//---------------------------------------------------------------------------------------------------------------
//
//  HAUD 2026.01.16
//
//  - ExternControl
//
//    - cyclic call to simulation class which handshakes the XtsStations in XtsTransport PLC
//
//---------------------------------------------------------------------------------------------------------------
PROGRAM MAIN_APP
VAR
  eInitXtsTransport   AT %I*    : e_progress;
  eInit                         : E_PROGRESS;   // application startup state info

  nProcess          : UINT;

  bNext             : BOOL := TRUE;
  bEnter            : BOOL := TRUE;
  bLeave            : BOOL := TRUE;

  tProcess          : ARRAY[1..MAX_PROCESS] OF TIME;

  eMtrState,
  eMsgState         : E_MESSAGE_STATE;
  eMtrProgress,
  eMsgProgress      : e_progress;
  stMsg             : ST_Message;
  //-------------------------------------------------------------------------------------------------------------
  tIdleWriteApplication   : TIME := T#5S;
  tIdleWriteMetric        : TIME := T#5S;
  tonIdleWriteApplication : Tc2_Standard.TON;
  tonIdleWriteMetric      : Tc2_Standard.TON;
  //-------------------------------------------------------------------------------------------------------------
END_VAR

//#################################################################################################################
// Local time; used for timestamps
//#################################################################################################################
GVL_MSG_XTS.fbLocalTime();
GVL_MSG_XTS.sLocalTime                                      := GVL_MSG_XTS.fbLocalTime.LocalTimeString;
GVL_MSG_XTS.dtLocalTime                                     := GVL_MSG_XTS.fbLocalTime.LocalTime;
//#################################################################################################################
//#################################################################################################################
//-----------------------------------------------------------------------------------------------------------------
//-----------------------------------------------------------------------------------------------------------------
// check for MAIN.eInit
//  - wait for fb_TransportUnit to be fully started up
//-----------------------------------------------------------------------------------------------------------------
IF NOT (eInitXtsTransport = E_PROGRESS.PROGRESS_DONE) THEN eInit   := E_PROGRESS.PROGRESS_INVALID; RETURN; END_IF
//-----------------------------------------------------------------------------------------------------------------
//-----------------------------------------------------------------------------------------------------------------
//-----------------------------------------------------------------------------------------------------------------
// /assign dataflow
//-----------------------------------------------------------------------------------------------------------------
FOR nProcess := 1 TO MAX_PROCESS
DO
  GVL_APPLICATION.Simulation[nProcess].ProcessId            := nProcess;
  GVL_APPLICATION.Simulation[nProcess].StationCtrl          := ADR(GVL_XTS.StationCtrl);
  GVL_APPLICATION.Simulation[nProcess].StationState         := ADR(GVL_XTS.StationState);

  GVL_APPLICATION.Simulation[nProcess].ProcessTime          := tProcess[nProcess];
  GVL_APPLICATION.Simulation[nProcess].MessageLevel         := GVL_MSG_XTS.MessageLevel;
END_FOR
//-----------------------------------------------------------------------------------------------------------------
//-----------------------------------------------------------------------------------------------------------------
Init();
//-----------------------------------------------------------------------------------------------------------------
//-----------------------------------------------------------------------------------------------------------------
// react to operation modes
//-----------------------------------------------------------------------------------------------------------------
//-----------------------------------------------------------------------------------------------------------------
CASE GVL_XTS.XtsTransportCtrl.Cmd
OF
  E_XTS_TRANSPORT_CTRL.CMD_INIT,
  E_XTS_TRANSPORT_CTRL.CMD_GROUP_CLEAR:

    FOR nProcess := 1 TO MAX_PROCESS
    DO
      GVL_APPLICATION.Simulation[nProcess].Init(); // clearing of XtsStations and Simulation
    END_FOR
END_CASE

CASE (GVL_XTS.XtsTransportState.State MOD E_PROGRESS.PROGRESS_DONE)
OF
  E_XTS_TRANSPORT_STATE.TRANSPORT_INIT,
  E_XTS_TRANSPORT_STATE.TRANSPORT_GROUP_CLEAR:
    FOR nProcess := 1 TO MAX_PROCESS
    DO
      GVL_APPLICATION.Simulation[nProcess].Disable(); // switch off XtsStations and clear Simulation

      GVL_APPLICATION.Simulation[nProcess].EnableProcess    := 0;
      GVL_APPLICATION.Simulation[nProcess].MoverEnter       := FALSE;
      GVL_APPLICATION.Simulation[nProcess].MoverOut         := FALSE;

      GVL_APPLICATION.Simulation[nProcess].Cycle();
    END_FOR

  E_XTS_TRANSPORT_STATE.TRANSPORT_START,
  E_XTS_TRANSPORT_STATE.TRANSPORT_RESTART:

    FOR nProcess := 1 TO MAX_PROCESS
    DO
      GVL_APPLICATION.Simulation[nProcess].Next(bNext);
      GVL_APPLICATION.Simulation[nProcess].Cycle();
    END_FOR
ELSE
  CASE (GVL_XTS.XtsTransportState.State MOD E_PROGRESS.PROGRESS_WORKING)
  OF
  E_XTS_TRANSPORT_STATE.TRANSPORT_START,
  E_XTS_TRANSPORT_STATE.TRANSPORT_RESTART:
    FOR nProcess := 1 TO MAX_PROCESS
    DO
      IF (GVL_APPLICATION.Simulation[nProcess].StationCount > 0)
      THEN
        GVL_APPLICATION.Simulation[nProcess].EnableProcess  := TO_DWORD(EXPT(2,GVL_APPLICATION.Simulation[nProcess].StationCount))-1;
        GVL_APPLICATION.Simulation[nProcess].MoverEnter     := TRUE;
        GVL_APPLICATION.Simulation[nProcess].MoverOut       := TRUE;

      END_IF

      GVL_APPLICATION.Simulation[nProcess].Next(bNext);
      GVL_APPLICATION.Simulation[nProcess].Cycle();
    END_FOR
  END_CASE
END_CASE
//-----------------------------------------------------------------------------------------------------------------
//-----------------------------------------------------------------------------------------------------------------
//#################################################################################################################
// /logging
//#################################################################################################################
GVL_MSG_XTS.ApplicationMessageData.Ctrl                         REF= GVL_MSG_XTS.ApplicationMessageCtrl;
GVL_MSG_XTS.ApplicationMessageData.State                        REF= GVL_MSG_XTS.ApplicationMessageState;

GVL_MSG_XTS.ApplicationMessageData.MessageIndex                 REF= GVL_MSG_XTS.MessageApplicationIndex;
GVL_MSG_XTS.ApplicationMessageData.ErrorIndex                   REF= GVL_MSG_XTS.MessageApplicationError;

GVL_MSG_XTS.ApplicationMessageData.DirRoot                      :=   ADR(GVL_MSG_XTS.LOG_DIR);
GVL_MSG_XTS.ApplicationMessageData.FileRoot                     :=   ADR(GVL_MSG_XTS.LOG_FILE_APP);
GVL_MSG_XTS.ApplicationMessageData.MsgList                      :=   ADR(GVL_MSG_XTS.ApplicationMessages);
GVL_MSG_XTS.ApplicationMessageData.LocalTime                    :=   ADR(GVL_MSG_XTS.dtLocalTime);

GVL_MSG_XTS.ApplicationMessageData();

eMsgState                                   := f_GetState   (GVL_MSG_XTS.ApplicationMessageState.State);
eMsgProgress                                := f_GetProgress(GVL_MSG_XTS.ApplicationMessageState.State);


CASE eMsgState
OF
  E_MESSAGE_STATE.MSG_STATE_NULL:
    CASE eMsgProgress
    OF
      E_PROGRESS.PROGRESS_INVALID:
        IF (GVL_MSG_XTS.MessageApplicationIndex > GVL_MSG_XTS.MAX_MESSAGE/100) OR
           (GVL_MSG_XTS.MessageApplicationError > 0)
        THEN
          GVL_MSG_XTS.ApplicationMessageCtrl.Cmd  := E_MESSAGE_CTRL.MSG_CTRL_WRITE;
        ELSE
          tonIdleWriteApplication(IN := TRUE, PT:= tIdleWriteApplication);
          IF (tonIdleWriteApplication.Q)
          THEN
            GVL_MSG_XTS.TransportMessageCtrl.Cmd    := E_MESSAGE_CTRL.MSG_CTRL_WRITE;
          END_IF
        END_IF
    END_CASE

  E_MESSAGE_STATE.MSG_STATE_WRITE:
    CASE eMsgProgress
    OF
      E_PROGRESS.PROGRESS_ERROR,
      E_PROGRESS.PROGRESS_DONE:
        tonIdleWriteApplication(IN := FALSE, PT:= tIdleWriteApplication);
        GVL_MSG_XTS.ApplicationMessageCtrl.Cmd    := E_MESSAGE_CTRL.MSG_CTRL_NULL;
    END_CASE

ELSE
    CASE eMsgProgress
    OF
      E_PROGRESS.PROGRESS_DONE:
        GVL_MSG_XTS.ApplicationMessageCtrl.Cmd    := E_MESSAGE_CTRL.MSG_CTRL_NULL;
    END_CASE
END_CASE
//#################################################################################################################
// logging/
//#################################################################################################################
//#################################################################################################################
//  /Transport Metrics
//#################################################################################################################
GVL_MSG_XTS.MetricsMessageData.Ctrl                             REF= GVL_MSG_XTS.MetricsMessageCtrl;
GVL_MSG_XTS.MetricsMessageData.State                            REF= GVL_MSG_XTS.MetricsMessageState;

GVL_MSG_XTS.MetricsMessageData.MessageIndex                     REF= GVL_MSG_XTS.MessageMetricsIndex;
GVL_MSG_XTS.MetricsMessageData.ErrorIndex                       REF= GVL_MSG_XTS.MessageMetricsError;

GVL_MSG_XTS.MetricsMessageData.DirRoot                          :=   ADR(GVL_MSG_XTS.LOG_DIR);
GVL_MSG_XTS.MetricsMessageData.FileRoot                         :=   ADR(GVL_MSG_XTS.LOG_FILE_METRIC);
GVL_MSG_XTS.MetricsMessageData.MsgList                          :=   ADR(GVL_MSG_XTS.MetricsMessages);
GVL_MSG_XTS.MetricsMessageData.LocalTime                        :=   ADR(GVL_MSG_XTS.dtLocalTime);

GVL_MSG_XTS.MetricsMessageData();

eMtrState                                   := f_GetState   (GVL_MSG_XTS.MetricsMessageState.State);
eMtrProgress                                := f_GetProgress(GVL_MSG_XTS.MetricsMessageState.State);

CASE eMtrState
OF
  E_MESSAGE_STATE.MSG_STATE_NULL:
    CASE eMtrProgress
    OF
      E_PROGRESS.PROGRESS_INVALID:
        IF (GVL_MSG_XTS.MessageMetricsIndex > GVL_MSG_XTS.MAX_MESSAGE/100) OR
           (GVL_MSG_XTS.MessageMetricsError > 0)
        THEN
          GVL_MSG_XTS.MetricsMessageCtrl.Cmd      := E_MESSAGE_CTRL.MSG_CTRL_WRITE;
        ELSE
          tonIdleWriteMetric(IN := TRUE, PT:= tIdleWriteMetric);
          IF (tonIdleWriteMetric.Q)
          THEN
            GVL_MSG_XTS.TransportMessageCtrl.Cmd    := E_MESSAGE_CTRL.MSG_CTRL_WRITE;
          END_IF
        END_IF
    END_CASE

  E_MESSAGE_STATE.MSG_STATE_WRITE:
    CASE eMtrProgress
    OF
      E_PROGRESS.PROGRESS_ERROR,
      E_PROGRESS.PROGRESS_DONE:
        tonIdleWriteMetric(IN := FALSE, PT:= tIdleWriteMetric);
        GVL_MSG_XTS.MetricsMessageCtrl.Cmd        := E_MESSAGE_CTRL.MSG_CTRL_NULL;
    END_CASE
ELSE
    CASE eMtrProgress
    OF
      E_PROGRESS.PROGRESS_DONE:
        GVL_MSG_XTS.MetricsMessageCtrl.Cmd        := E_MESSAGE_CTRL.MSG_CTRL_NULL;
    END_CASE
END_CASE
//#################################################################################################################
//  Transport Metrics/
//#################################################################################################################
//#################################################################################################################
//#################################################################################################################

ACTION Init:
CASE eInit
OF
  E_PROGRESS.PROGRESS_INVALID:          // startup procedure for your application
    GVL_MSG_XTS.TransportMessageCtrl.Cmd                  := E_MESSAGE_CTRL.MSG_CTRL_NULL;
    GVL_MSG_XTS.MetricsMessageCtrl.Cmd                    := E_MESSAGE_CTRL.MSG_CTRL_NULL;

    FOR nProcess := 1 TO MAX_PROCESS
    DO
      GVL_MSG_XTS.MessageLevelProcess[nProcess]           := GVL_MSG_XTS.MessageLevel;

      GVL_APPLICATION.Simulation[nProcess].MessageLevel   := GVL_MSG_XTS.MessageLevelProcess[nProcess];
    END_FOR
    eInit                               := E_PROGRESS.PROGRESS_INIT;


  E_PROGRESS.PROGRESS_INIT:
      nProcess                                        := 1;
      tProcess[nProcess]                              := T#750MS;

      GVL_APPLICATION.Simulation[nProcess].StationFirst  := 1;
      GVL_APPLICATION.Simulation[nProcess].StationLast   := 16;

      GVL_APPLICATION.Simulation[nProcess].TargetFirst   := 20;
      GVL_APPLICATION.Simulation[nProcess].TargetLast    := 35;
      GVL_APPLICATION.Simulation[nProcess].TargetMask    := 2#0001; // mask for target station

      GVL_APPLICATION.Simulation[nProcess].CheckRangeLow := 1750.0;
      GVL_APPLICATION.Simulation[nProcess].CheckRangeHigh:= 2100.0;

      //---------------------------------------------------------

      // 2

      //---------------------------------------------------------
      nProcess                                        := 3;
      tProcess[nProcess]                              := T#1250MS;

      GVL_APPLICATION.Simulation[nProcess].StationFirst  := 20;
      GVL_APPLICATION.Simulation[nProcess].StationLast   := 35;

      GVL_APPLICATION.Simulation[nProcess].TargetFirst   := 37;
      GVL_APPLICATION.Simulation[nProcess].TargetLast    := 37;
      GVL_APPLICATION.Simulation[nProcess].TargetMask    := 2#0001; // mask for target station

      GVL_APPLICATION.Simulation[nProcess].CheckRangeLow := 4500.0;
      GVL_APPLICATION.Simulation[nProcess].CheckRangeHigh:= 5100.0;

      //---------------------------------------------------------
      nProcess                                        := 4;
      tProcess[nProcess]                              := T#0MS;

      GVL_APPLICATION.Simulation[nProcess].StationFirst  := 37;
      GVL_APPLICATION.Simulation[nProcess].StationLast   := 37;

      GVL_APPLICATION.Simulation[nProcess].TargetFirst   := 45;
      GVL_APPLICATION.Simulation[nProcess].TargetLast    := 52;
      GVL_APPLICATION.Simulation[nProcess].TargetMask    := 2#0001; // mask for target station

      GVL_APPLICATION.Simulation[nProcess].CheckRangeLow := 7450.0;
      GVL_APPLICATION.Simulation[nProcess].CheckRangeHigh:= 7600.0;

      //---------------------------------------------------------
      nProcess                                        := 5;
      tProcess[nProcess]                              := T#500MS;

      GVL_APPLICATION.Simulation[nProcess].StationFirst  := 45;
      GVL_APPLICATION.Simulation[nProcess].StationLast   := 52;

      GVL_APPLICATION.Simulation[nProcess].TargetFirst   := 58;
      GVL_APPLICATION.Simulation[nProcess].TargetLast    := 69;
      GVL_APPLICATION.Simulation[nProcess].TargetMask    := 2#0001; // mask for target station

      GVL_APPLICATION.Simulation[nProcess].CheckRangeLow := 6600.0;
      GVL_APPLICATION.Simulation[nProcess].CheckRangeHigh:= 8350.0;

      //---------------------------------------------------------
      nProcess                                        := 6;
      tProcess[nProcess]                              := T#500MS;

      GVL_APPLICATION.Simulation[nProcess].StationFirst  := 58;
      GVL_APPLICATION.Simulation[nProcess].StationLast   := 69;

      GVL_APPLICATION.Simulation[nProcess].TargetFirst   := 70;
      GVL_APPLICATION.Simulation[nProcess].TargetLast    := 81;
      GVL_APPLICATION.Simulation[nProcess].TargetMask    := 2#0001; // mask for target station

      GVL_APPLICATION.Simulation[nProcess].CheckRangeLow := 8750.0;
      GVL_APPLICATION.Simulation[nProcess].CheckRangeHigh:= 9600.0;

      //---------------------------------------------------------
      nProcess                                        := 7;
      tProcess[nProcess]                              := T#500MS;

      GVL_APPLICATION.Simulation[nProcess].StationFirst  := 70;
      GVL_APPLICATION.Simulation[nProcess].StationLast   := 81;

      GVL_APPLICATION.Simulation[nProcess].TargetFirst   := 82;
      GVL_APPLICATION.Simulation[nProcess].TargetLast    := 91;
      GVL_APPLICATION.Simulation[nProcess].TargetMask    := 2#0001; // mask for target station

      GVL_APPLICATION.Simulation[nProcess].CheckRangeLow := 10900.0;
      GVL_APPLICATION.Simulation[nProcess].CheckRangeHigh:= 11600.0;

      //---------------------------------------------------------
      nProcess                                        := 8;
      tProcess[nProcess]                              := T#500MS;

      GVL_APPLICATION.Simulation[nProcess].StationFirst  := 82;
      GVL_APPLICATION.Simulation[nProcess].StationLast   := 91;

      GVL_APPLICATION.Simulation[nProcess].TargetFirst   := 92;
      GVL_APPLICATION.Simulation[nProcess].TargetLast    := 99;
      GVL_APPLICATION.Simulation[nProcess].TargetMask    := 2#0001; // mask for target station

      GVL_APPLICATION.Simulation[nProcess].CheckRangeLow := 12550.0;
      GVL_APPLICATION.Simulation[nProcess].CheckRangeHigh:= 12900.0;

      //---------------------------------------------------------
      nProcess                                        := 9;
      tProcess[nProcess]                              := T#500MS;

      GVL_APPLICATION.Simulation[nProcess].StationFirst  := 92;
      GVL_APPLICATION.Simulation[nProcess].StationLast   := 99;

      GVL_APPLICATION.Simulation[nProcess].TargetFirst   := 118;
      GVL_APPLICATION.Simulation[nProcess].TargetLast    := 118;
      GVL_APPLICATION.Simulation[nProcess].TargetMask    := 2#0001; // mask for target station

      GVL_APPLICATION.Simulation[nProcess].CheckRangeLow := 13600.0;
      GVL_APPLICATION.Simulation[nProcess].CheckRangeHigh:= 14600.0;

      //---------------------------------------------------------
      nProcess                                        := 12;
      tProcess[nProcess]                              := T#600MS;

      GVL_APPLICATION.Simulation[nProcess].StationFirst  := 110;
      GVL_APPLICATION.Simulation[nProcess].StationLast   := 117;

      GVL_APPLICATION.Simulation[nProcess].TargetFirst   := 134;
      GVL_APPLICATION.Simulation[nProcess].TargetLast    := 147;
      GVL_APPLICATION.Simulation[nProcess].TargetMask    := 2#0001; // mask for target station

      GVL_APPLICATION.Simulation[nProcess].CheckRangeLow := 16500.0;
      GVL_APPLICATION.Simulation[nProcess].CheckRangeHigh:= 17100.0;

      //---------------------------------------------------------
      nProcess                                        := 13;
      tProcess[nProcess]                              := T#00MS;

      GVL_APPLICATION.Simulation[nProcess].StationFirst  := 118;
      GVL_APPLICATION.Simulation[nProcess].StationLast   := 118;

      GVL_APPLICATION.Simulation[nProcess].TargetFirst   := 119;
      GVL_APPLICATION.Simulation[nProcess].TargetLast    := 119;
      GVL_APPLICATION.Simulation[nProcess].TargetMask    := 2#0001; // mask for target station

      GVL_APPLICATION.Simulation[nProcess].CheckRangeLow := 15400.0;
      GVL_APPLICATION.Simulation[nProcess].CheckRangeHigh:= 15600.0;

      //---------------------------------------------------------
      nProcess                                        := 14;
      tProcess[nProcess]                              := T#0MS;

      GVL_APPLICATION.Simulation[nProcess].StationFirst  := 119;
      GVL_APPLICATION.Simulation[nProcess].StationLast   := 119;

      GVL_APPLICATION.Simulation[nProcess].TargetFirst   := 110;
      GVL_APPLICATION.Simulation[nProcess].TargetLast    := 117;
      GVL_APPLICATION.Simulation[nProcess].TargetMask    := 2#0001; // mask for target station

      GVL_APPLICATION.Simulation[nProcess].CheckRangeLow := 15750.0;
      GVL_APPLICATION.Simulation[nProcess].CheckRangeHigh:= 16250.0;

      //---------------------------------------------------------


      //---------------------------------------------------------
      nProcess                                        := 16;
      tProcess[nProcess]                              := T#750MS;

      GVL_APPLICATION.Simulation[nProcess].StationFirst  := 134;
      GVL_APPLICATION.Simulation[nProcess].StationLast   := 147;

      GVL_APPLICATION.Simulation[nProcess].TargetFirst   := 148;
      GVL_APPLICATION.Simulation[nProcess].TargetLast    := 148;
      GVL_APPLICATION.Simulation[nProcess].TargetMask    := 2#0001; // mask for target station

      GVL_APPLICATION.Simulation[nProcess].CheckRangeLow := 18500.0;
      GVL_APPLICATION.Simulation[nProcess].CheckRangeHigh:= 19600.0;

      //---------------------------------------------------------
      nProcess                                        := 17;
      tProcess[nProcess]                              := T#0MS;

      GVL_APPLICATION.Simulation[nProcess].StationFirst  := 148;
      GVL_APPLICATION.Simulation[nProcess].StationLast   := 148;

      GVL_APPLICATION.Simulation[nProcess].TargetFirst   := 149;
      GVL_APPLICATION.Simulation[nProcess].TargetLast    := 149;
      GVL_APPLICATION.Simulation[nProcess].TargetMask    := 2#0001; // mask for target station

      GVL_APPLICATION.Simulation[nProcess].CheckRangeLow := 21750.0;
      GVL_APPLICATION.Simulation[nProcess].CheckRangeHigh:= 22100.0;

      //---------------------------------------------------------
      nProcess                                        := 18;
      tProcess[nProcess]                              := T#0MS;

      GVL_APPLICATION.Simulation[nProcess].StationFirst  := 149;
      GVL_APPLICATION.Simulation[nProcess].StationLast   := 149;

      GVL_APPLICATION.Simulation[nProcess].TargetFirst   := 150;
      GVL_APPLICATION.Simulation[nProcess].TargetLast    := 150;
      GVL_APPLICATION.Simulation[nProcess].TargetMask    := 2#0001; // mask for target station

      GVL_APPLICATION.Simulation[nProcess].CheckRangeLow := 22450.0;
      GVL_APPLICATION.Simulation[nProcess].CheckRangeHigh:= 22700.0;

      //---------------------------------------------------------
      nProcess                                        := 19;
      tProcess[nProcess]                              := T#0MS;

      GVL_APPLICATION.Simulation[nProcess].StationFirst  := 150;
      GVL_APPLICATION.Simulation[nProcess].StationLast   := 150;

      GVL_APPLICATION.Simulation[nProcess].TargetFirst   := 1;
      GVL_APPLICATION.Simulation[nProcess].TargetLast    := 16;
      GVL_APPLICATION.Simulation[nProcess].TargetMask    := 2#0001; // mask for target station

      GVL_APPLICATION.Simulation[nProcess].CheckRangeLow := 500.0;
      GVL_APPLICATION.Simulation[nProcess].CheckRangeHigh:= 2100.0;

    eInit                                                 := E_PROGRESS.PROGRESS_BUSY;

  E_PROGRESS.PROGRESS_BUSY:
    GVL_MSG_XTS.TransportMessageCtrl.Cmd                  := E_MESSAGE_CTRL.MSG_CTRL_INIT;
    GVL_MSG_XTS.MetricsMessageCtrl.Cmd                    := E_MESSAGE_CTRL.MSG_CTRL_INIT;
    eInit                                                 := E_PROGRESS.PROGRESS_PREPARE;

  E_PROGRESS.PROGRESS_PREPARE:
    eInit                                                 := E_PROGRESS.PROGRESS_DONE;

END_CASE
END_ACTION

END_PROGRAM

(* stored: Version 1.1.0.1
   POU MAIN_APP: Id {aed82ec5-7c0f-4ed8-9d95-00008ab7747f}, SpecialFunc None
   Action Init: Id {69838e0d-19cf-48fe-8b42-ee1af1eba2b6} *)
